TYPE ST_MESSAGE_STATE :
STRUCT
  State         : E_MESSAGE_STATE;  // as always... combined value of Cmd equivalent and e_progress
END_STRUCT
END_TYPE

(* stored: Version 1.1.0.1, ProductVersion 3.1.4026.18
   DUT ST_MESSAGE_STATE: Id {a5dc31e5-43d2-4fa7-94ef-ebe6543ff6ef} *)
